// TIA Portal V19 export
TYPE "Decoiler_Manager"
   STRUCT
      IsOutLine : Bool;
      IsInLine : Bool;
      EmptiyngConfirmed : Bool;
      ModePneumaticBraking : Bool;
      TotalBrakeOpeningAttempt : Bool;
      Feed : "SpeedMachine_CIn_Manager";
      Coupling { S7_SetPoint := 'True'} : "ValveMachine_Manager";
      Jaws : "ValveMachine_Manager";
      SnubberLift { S7_SetPoint := 'True'} : "ValveMachine_Manager";
      SnubberRoll { S7_SetPoint := 'True'} : "ValveMachine_Manager";
   END_STRUCT;
END_TYPE
